{attribute 'GeneratedUsingTerminal: EL9560-0000-0016'}
{attribute addProperty BoxType "EL9560-0000-0016"}
{attribute addProperty Id "Power_OKAT %I*BOOL1"}
{attribute addProperty CRC "1151167157"}
{attribute addProperty Size "1"}
TYPE Status_Uo_449D6AB5 :
STRUCT
	{attribute addProperty Name "Power_OK"}
	Power_OK AT %I* : BOOL;
END_STRUCT
END_TYPE

(* stored: Version 1.2.0.0, ProductVersion 3.1.4024.9
   DUT Status_Uo_449D6AB5: Id {586d6428-59c3-499e-82e1-14335c07f40e} *)
